// TIA Portal V19 export
FUNCTION_BLOCK "F_Zone25_FB"   // FB169, F_LAD
TITLE = SAFETY ZONE 25 - AREA 03 (PAREGGIAMENTO)
// stored: Access Published
   VAR
      D25 : "Door_FB";
      D27 : "Door_FB";
      FNS : "ForceNormalStop";
      F_Sinamics_Rulliera_1 : "FDevice_Sinamics_FB";
      F_Sinamics_Rulliera_2 : "FDevice_Sinamics_FB";
      F_Sinamics_PareggiatoreTesta : "FDevice_Sinamics_FB";
      F_Sinamics_PareggiatoreCoda : "FDevice_Sinamics_FB";
      F_Sinamics_ManipolatoreTesta : "FDevice_Sinamics_FB";
      F_Sinamics_ManipolatoreCoda : "FDevice_Sinamics_FB";
      F_Contactor_Valvole_Pareggiatore_Testa : "FDevice_Contactor_FB";
      F_Contactor_Valvole_Pareggiatore_Coda : "FDevice_Contactor_FB";
      F_Contactor_HU_CYTROPAC_STO { ExternalAccessible := 'False'; ExternalVisible := 'False'; ExternalWritable := 'False'} : "FDevice_Contactor_FB";
   END_VAR
   VAR_TEMP
      DoorNormalStop : Bool;
      DoorSafeStop : Bool;
      Door_Ok : Bool;
      FDBK : Bool;
   END_VAR
BEGIN

REGION Network 1: < < < < < < < < < < DOOR > > > > > > > > > >
END_REGION

REGION Network 2: Zone Entry enable
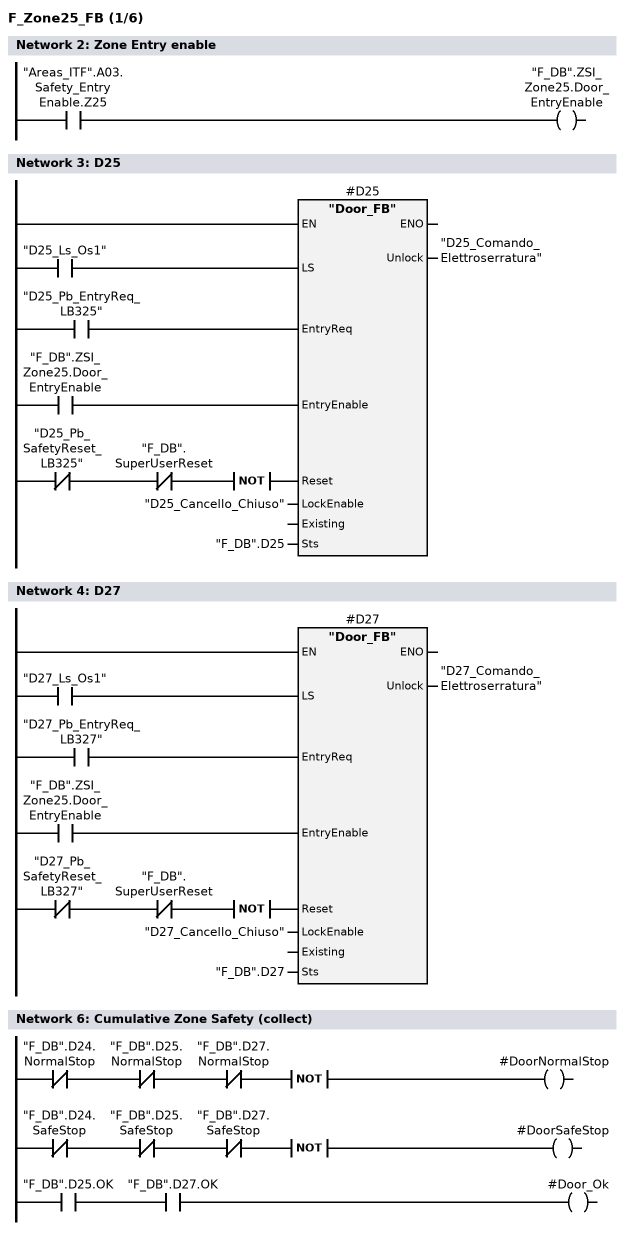
   RUNG wire#powerrail
      Contact( "Areas_ITF".A03.Safety_EntryEnable.Z25 )
      Coil( "F_DB".ZSI_Zone25.Door_EntryEnable )
   END_RUNG
   // the same network as SCL:
   "F_DB".ZSI_Zone25.Door_EntryEnable := "Areas_ITF".A03.Safety_EntryEnable.Z25;
END_REGION

REGION Network 3: D25
   RUNG wire#powerrail
      #D25(LS := wire#w1, EntryReq := wire#w2, EntryEnable := wire#w3, Reset := wire#w4, LockEnable := "D25_Cancello_Chiuso", Existing :=, Sts := "F_DB".D25, Unlock => "D25_Comando_Elettroserratura")
   END_RUNG
   RUNG wire#powerrail
      Contact( "D25_Ls_Os1" )
   END_RUNG wire#w1
   RUNG wire#powerrail
      Contact( "D25_Pb_EntryReq_LB325" )
   END_RUNG wire#w2
   RUNG wire#powerrail
      Contact( "F_DB".ZSI_Zone25.Door_EntryEnable )
   END_RUNG wire#w3
   RUNG wire#powerrail
      I_Contact( "D25_Pb_SafetyReset_LB325" )
      I_Contact( "F_DB".SuperUserReset )
      Not()
   END_RUNG wire#w4
   // the same network as SCL:
   #D25(LS := "D25_Ls_Os1",   // "Door_FB"
        EntryReq := "D25_Pb_EntryReq_LB325",
        EntryEnable := "F_DB".ZSI_Zone25.Door_EntryEnable,
        Reset := NOT (NOT "D25_Pb_SafetyReset_LB325" AND NOT "F_DB".SuperUserReset),
        LockEnable := "D25_Cancello_Chiuso",
        Sts := "F_DB".D25,
        Unlock => "D25_Comando_Elettroserratura");
END_REGION

REGION Network 4: D27
   RUNG wire#powerrail
      #D27(LS := wire#w1, EntryReq := wire#w2, EntryEnable := wire#w3, Reset := wire#w4, LockEnable := "D27_Cancello_Chiuso", Existing :=, Sts := "F_DB".D27, Unlock => "D27_Comando_Elettroserratura")
   END_RUNG
   RUNG wire#powerrail
      Contact( "D27_Ls_Os1" )
   END_RUNG wire#w1
   RUNG wire#powerrail
      Contact( "D27_Pb_EntryReq_LB327" )
   END_RUNG wire#w2
   RUNG wire#powerrail
      Contact( "F_DB".ZSI_Zone25.Door_EntryEnable )
   END_RUNG wire#w3
   RUNG wire#powerrail
      I_Contact( "D27_Pb_SafetyReset_LB327" )
      I_Contact( "F_DB".SuperUserReset )
      Not()
   END_RUNG wire#w4
   // the same network as SCL:
   #D27(LS := "D27_Ls_Os1",   // "Door_FB"
        EntryReq := "D27_Pb_EntryReq_LB327",
        EntryEnable := "F_DB".ZSI_Zone25.Door_EntryEnable,
        Reset := NOT (NOT "D27_Pb_SafetyReset_LB327" AND NOT "F_DB".SuperUserReset),
        LockEnable := "D27_Cancello_Chiuso",
        Sts := "F_DB".D27,
        Unlock => "D27_Comando_Elettroserratura");
END_REGION

REGION Network 5: < < < < < < < < < < ZONE SAFETY INTERFACE > > > > > > > > > >
END_REGION

REGION Network 6: Cumulative Zone Safety (collect)
   RUNG wire#powerrail
      I_Contact( "F_DB".D24.NormalStop )
      I_Contact( "F_DB".D25.NormalStop )
      I_Contact( "F_DB".D27.NormalStop )
      Not()
      Coil( #DoorNormalStop )
   END_RUNG
   RUNG wire#powerrail
      I_Contact( "F_DB".D24.SafeStop )
      I_Contact( "F_DB".D25.SafeStop )
      I_Contact( "F_DB".D27.SafeStop )
      Not()
      Coil( #DoorSafeStop )
   END_RUNG
   RUNG wire#powerrail
      Contact( "F_DB".D25.OK )
      Contact( "F_DB".D27.OK )
      Coil( #Door_Ok )
   END_RUNG
   // the same network as SCL:
   #DoorNormalStop := NOT (NOT "F_DB".D24.NormalStop AND NOT "F_DB".D25.NormalStop AND NOT "F_DB".D27.NormalStop);
   #DoorSafeStop := NOT (NOT "F_DB".D24.SafeStop AND NOT "F_DB".D25.SafeStop AND NOT "F_DB".D27.SafeStop);
   #Door_Ok := "F_DB".D25.OK AND "F_DB".D27.OK;
END_REGION

REGION Network 7: Zone must stay in Normal Stop During Restart
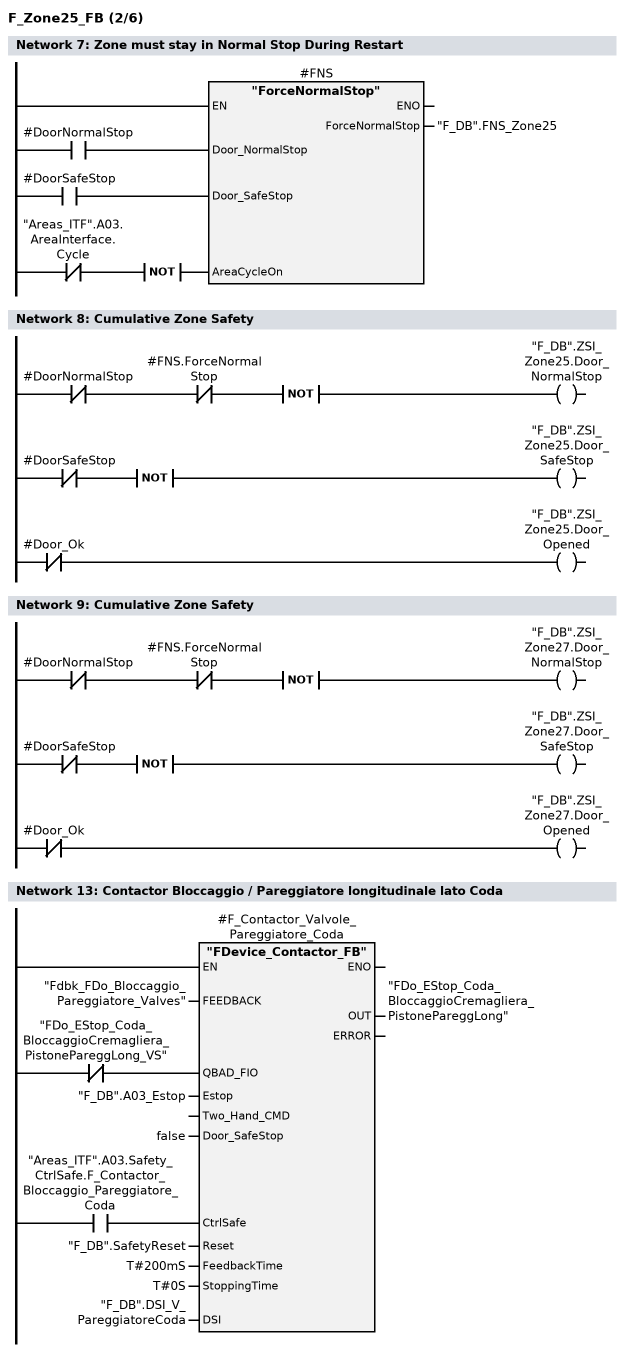
   RUNG wire#powerrail
      #FNS(Door_NormalStop := wire#w1, Door_SafeStop := wire#w2, AreaCycleOn := wire#w3, ForceNormalStop => "F_DB".FNS_Zone25)
   END_RUNG
   RUNG wire#powerrail
      Contact( #DoorNormalStop )
   END_RUNG wire#w1
   RUNG wire#powerrail
      Contact( #DoorSafeStop )
   END_RUNG wire#w2
   RUNG wire#powerrail
      I_Contact( "Areas_ITF".A03.AreaInterface.Cycle )
      Not()
   END_RUNG wire#w3
   // the same network as SCL:
   #FNS(Door_NormalStop := #DoorNormalStop,   // "ForceNormalStop"
        Door_SafeStop := #DoorSafeStop,
        AreaCycleOn := NOT (NOT "Areas_ITF".A03.AreaInterface.Cycle),
        ForceNormalStop => "F_DB".FNS_Zone25);
END_REGION

REGION Network 8: Cumulative Zone Safety
   RUNG wire#powerrail
      I_Contact( #DoorNormalStop )
      I_Contact( #FNS.ForceNormalStop )
      Not()
      Coil( "F_DB".ZSI_Zone25.Door_NormalStop )
   END_RUNG
   RUNG wire#powerrail
      I_Contact( #DoorSafeStop )
      Not()
      Coil( "F_DB".ZSI_Zone25.Door_SafeStop )
   END_RUNG
   RUNG wire#powerrail
      I_Contact( #Door_Ok )
      Coil( "F_DB".ZSI_Zone25.Door_Opened )
   END_RUNG
   // the same network as SCL:
   "F_DB".ZSI_Zone25.Door_NormalStop := NOT (NOT #DoorNormalStop AND NOT #FNS.ForceNormalStop);
   "F_DB".ZSI_Zone25.Door_SafeStop := NOT (NOT #DoorSafeStop);
   "F_DB".ZSI_Zone25.Door_Opened := NOT #Door_Ok;
END_REGION

REGION Network 9: Cumulative Zone Safety
   RUNG wire#powerrail
      I_Contact( #DoorNormalStop )
      I_Contact( #FNS.ForceNormalStop )
      Not()
      Coil( "F_DB".ZSI_Zone27.Door_NormalStop )
   END_RUNG
   RUNG wire#powerrail
      I_Contact( #DoorSafeStop )
      Not()
      Coil( "F_DB".ZSI_Zone27.Door_SafeStop )
   END_RUNG
   RUNG wire#powerrail
      I_Contact( #Door_Ok )
      Coil( "F_DB".ZSI_Zone27.Door_Opened )
   END_RUNG
   // the same network as SCL:
   "F_DB".ZSI_Zone27.Door_NormalStop := NOT (NOT #DoorNormalStop AND NOT #FNS.ForceNormalStop);
   "F_DB".ZSI_Zone27.Door_SafeStop := NOT (NOT #DoorSafeStop);
   "F_DB".ZSI_Zone27.Door_Opened := NOT #Door_Ok;
END_REGION

REGION Network 10: >
END_REGION

REGION Network 11: >
END_REGION

REGION Network 12: < < < < < < < < < < DEVICES SAFETY VALVES > > > > > > > > > >
END_REGION

REGION Network 13: Contactor Bloccaggio / Pareggiatore longitudinale lato Coda
   RUNG wire#powerrail
      #F_Contactor_Valvole_Pareggiatore_Coda(QBAD_FIO := wire#w1, CtrlSafe := wire#w2, FEEDBACK := "Fdbk_FDo_Bloccaggio_Pareggiatore_Valves", Estop := "F_DB".A03_Estop, Two_Hand_CMD :=, Door_SafeStop := false, Reset := "F_DB".SafetyReset, FeedbackTime := T#200mS, StoppingTime := T#0S, DSI := "F_DB".DSI_V_PareggiatoreCoda, OUT => "FDo_EStop_Coda_BloccaggioCremagliera_PistonePareggLong", ERROR =>)
   END_RUNG
   RUNG wire#powerrail
      I_Contact( "FDo_EStop_Coda_BloccaggioCremagliera_PistonePareggLong_VS" )
   END_RUNG wire#w1
   RUNG wire#powerrail
      Contact( "Areas_ITF".A03.Safety_CtrlSafe.F_Contactor_Bloccaggio_Pareggiatore_Coda )
   END_RUNG wire#w2
   // the same network as SCL:
   #F_Contactor_Valvole_Pareggiatore_Coda(FEEDBACK := "Fdbk_FDo_Bloccaggio_Pareggiatore_Valves",   // "FDevice_Contactor_FB"
                           QBAD_FIO := NOT "FDo_EStop_Coda_BloccaggioCremagliera_PistonePareggLong_VS",
                           Estop := "F_DB".A03_Estop,
                           Door_SafeStop := false,
                           CtrlSafe := "Areas_ITF".A03.Safety_CtrlSafe.F_Contactor_Bloccaggio_Pareggiatore_Coda,
                           Reset := "F_DB".SafetyReset,
                           FeedbackTime := T#200mS,
                           StoppingTime := T#0S,
                           DSI := "F_DB".DSI_V_PareggiatoreCoda,
                           OUT => "FDo_EStop_Coda_BloccaggioCremagliera_PistonePareggLong");
END_REGION

REGION Network 14: Contactor Bloccaggio lato testa
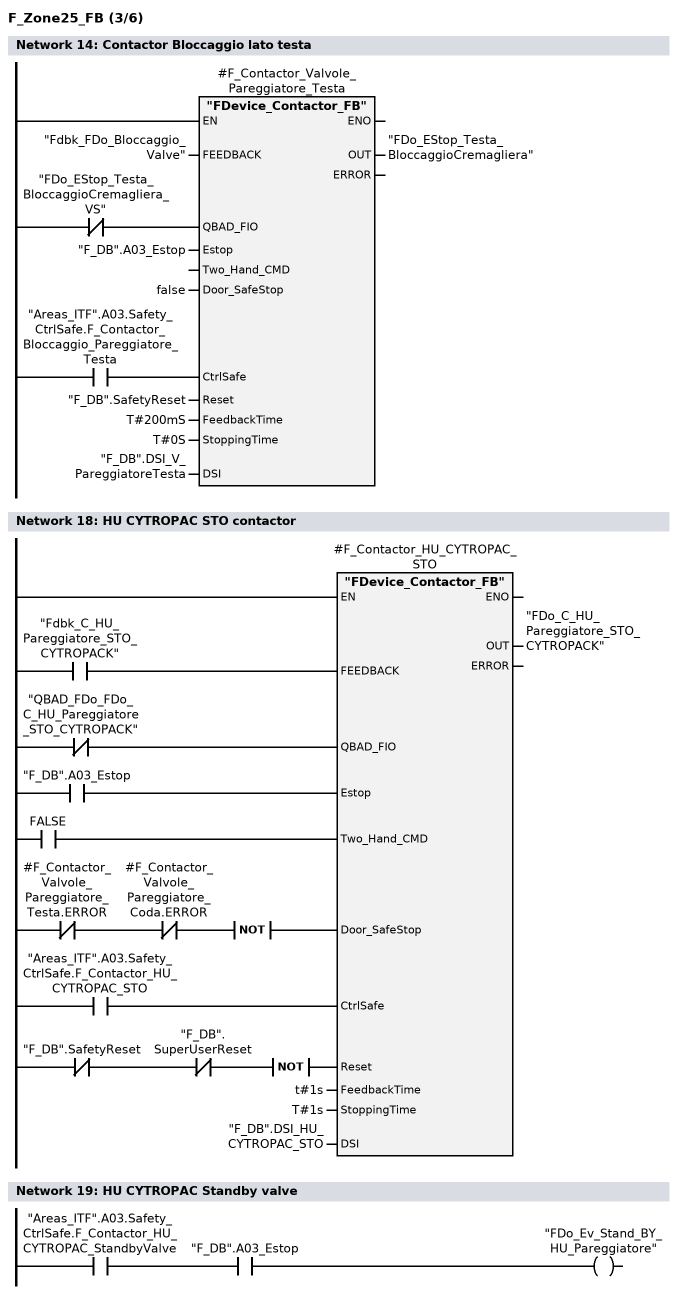
   RUNG wire#powerrail
      #F_Contactor_Valvole_Pareggiatore_Testa(QBAD_FIO := wire#w1, CtrlSafe := wire#w2, FEEDBACK := "Fdbk_FDo_Bloccaggio_Valve", Estop := "F_DB".A03_Estop, Two_Hand_CMD :=, Door_SafeStop := false, Reset := "F_DB".SafetyReset, FeedbackTime := T#200mS, StoppingTime := T#0S, DSI := "F_DB".DSI_V_PareggiatoreTesta, OUT => "FDo_EStop_Testa_BloccaggioCremagliera", ERROR =>)
   END_RUNG
   RUNG wire#powerrail
      I_Contact( "FDo_EStop_Testa_BloccaggioCremagliera_VS" )
   END_RUNG wire#w1
   RUNG wire#powerrail
      Contact( "Areas_ITF".A03.Safety_CtrlSafe.F_Contactor_Bloccaggio_Pareggiatore_Testa )
   END_RUNG wire#w2
   // the same network as SCL:
   #F_Contactor_Valvole_Pareggiatore_Testa(FEEDBACK := "Fdbk_FDo_Bloccaggio_Valve",   // "FDevice_Contactor_FB"
                           QBAD_FIO := NOT "FDo_EStop_Testa_BloccaggioCremagliera_VS",
                           Estop := "F_DB".A03_Estop,
                           Door_SafeStop := false,
                           CtrlSafe := "Areas_ITF".A03.Safety_CtrlSafe.F_Contactor_Bloccaggio_Pareggiatore_Testa,
                           Reset := "F_DB".SafetyReset,
                           FeedbackTime := T#200mS,
                           StoppingTime := T#0S,
                           DSI := "F_DB".DSI_V_PareggiatoreTesta,
                           OUT => "FDo_EStop_Testa_BloccaggioCremagliera");
END_REGION

REGION Network 15: >
END_REGION

REGION Network 16: >
END_REGION

REGION Network 17: < < < < < < < < < < DEVICES CONTACTORS > > > > > > > > > >
END_REGION

REGION Network 18: HU CYTROPAC STO contactor
   RUNG wire#powerrail
      #F_Contactor_HU_CYTROPAC_STO(FEEDBACK := wire#w1, QBAD_FIO := wire#w2, Estop := wire#w3, Two_Hand_CMD := wire#w4, Door_SafeStop := wire#w5, CtrlSafe := wire#w6, Reset := wire#w7, FeedbackTime := t#1s, StoppingTime := T#1s, DSI := "F_DB".DSI_HU_CYTROPAC_STO, OUT => "FDo_C_HU_Pareggiatore_STO_CYTROPACK", ERROR =>)
   END_RUNG
   RUNG wire#powerrail
      Contact( "Fdbk_C_HU_Pareggiatore_STO_CYTROPACK" )
   END_RUNG wire#w1
   RUNG wire#powerrail
      I_Contact( "QBAD_FDo_FDo_C_HU_Pareggiatore_STO_CYTROPACK" )
   END_RUNG wire#w2
   RUNG wire#powerrail
      Contact( "F_DB".A03_Estop )
   END_RUNG wire#w3
   RUNG wire#powerrail
      Contact( FALSE )
   END_RUNG wire#w4
   RUNG wire#powerrail
      I_Contact( #F_Contactor_Valvole_Pareggiatore_Testa.ERROR )
      I_Contact( #F_Contactor_Valvole_Pareggiatore_Coda.ERROR )
      Not()
   END_RUNG wire#w5
   RUNG wire#powerrail
      Contact( "Areas_ITF".A03.Safety_CtrlSafe.F_Contactor_HU_CYTROPAC_STO )
   END_RUNG wire#w6
   RUNG wire#powerrail
      I_Contact( "F_DB".SafetyReset )
      I_Contact( "F_DB".SuperUserReset )
      Not()
   END_RUNG wire#w7
   // the same network as SCL:
   #F_Contactor_HU_CYTROPAC_STO(FEEDBACK := "Fdbk_C_HU_Pareggiatore_STO_CYTROPACK",   // "FDevice_Contactor_FB"
                           QBAD_FIO := NOT "QBAD_FDo_FDo_C_HU_Pareggiatore_STO_CYTROPACK",
                           Estop := "F_DB".A03_Estop,
                           Two_Hand_CMD := FALSE,
                           Door_SafeStop := NOT (NOT #F_Contactor_Valvole_Pareggiatore_Testa.ERROR AND NOT #F_Contactor_Valvole_Pareggiatore_Coda.ERROR),
                           CtrlSafe := "Areas_ITF".A03.Safety_CtrlSafe.F_Contactor_HU_CYTROPAC_STO,
                           Reset := NOT (NOT "F_DB".SafetyReset AND NOT "F_DB".SuperUserReset),
                           FeedbackTime := t#1s,
                           StoppingTime := T#1s,
                           DSI := "F_DB".DSI_HU_CYTROPAC_STO,
                           OUT => "FDo_C_HU_Pareggiatore_STO_CYTROPACK");
END_REGION

REGION Network 19: HU CYTROPAC Standby valve
   RUNG wire#powerrail
      Contact( "Areas_ITF".A03.Safety_CtrlSafe.F_Contactor_HU_CYTROPAC_StandbyValve )
      Contact( "F_DB".A03_Estop )
      Coil( "FDo_Ev_Stand_BY_HU_Pareggiatore" )
   END_RUNG
   // the same network as SCL:
   "FDo_Ev_Stand_BY_HU_Pareggiatore" := "Areas_ITF".A03.Safety_CtrlSafe.F_Contactor_HU_CYTROPAC_StandbyValve AND "F_DB".A03_Estop;
END_REGION

REGION Network 20: >
END_REGION

REGION Network 21: >
END_REGION

REGION Network 22: < < < < < < < < < < DEVICES S120 > > > > > > > > > >
END_REGION

REGION Network 23: S120 - Ax Rulliera 1
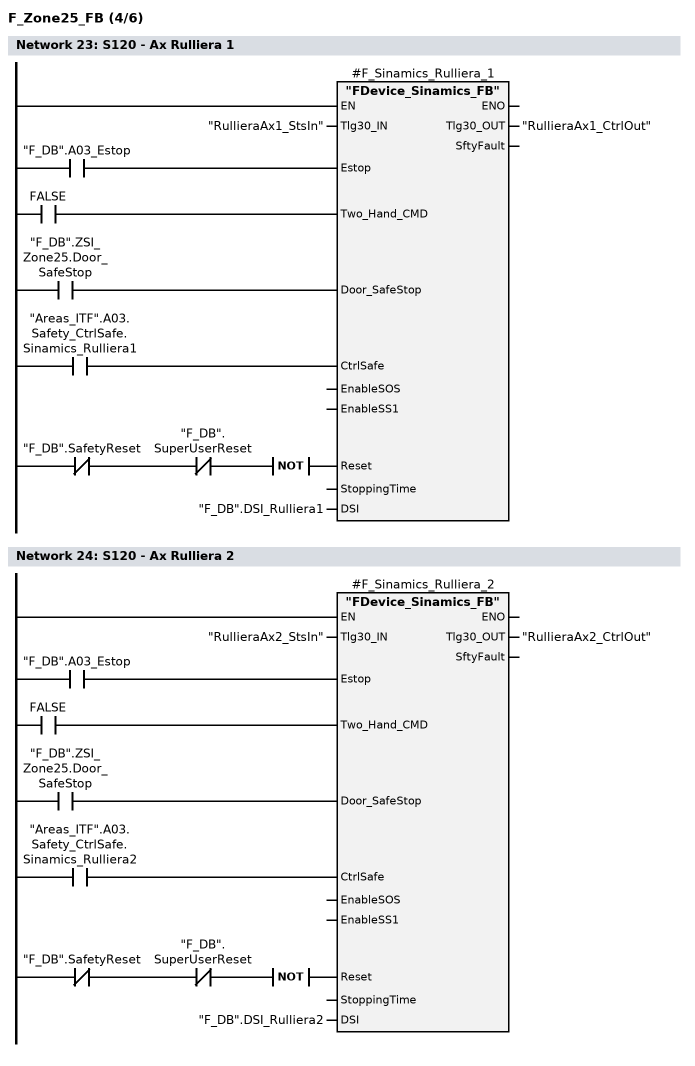
   RUNG wire#powerrail
      #F_Sinamics_Rulliera_1(Estop := wire#w1, Two_Hand_CMD := wire#w2, Door_SafeStop := wire#w3, CtrlSafe := wire#w4, Reset := wire#w5, Tlg30_IN := "RullieraAx1_StsIn", EnableSOS :=, EnableSS1 :=, StoppingTime :=, DSI := "F_DB".DSI_Rulliera1, Tlg30_OUT => "RullieraAx1_CtrlOut", SftyFault =>)
   END_RUNG
   RUNG wire#powerrail
      Contact( "F_DB".A03_Estop )
   END_RUNG wire#w1
   RUNG wire#powerrail
      Contact( FALSE )
   END_RUNG wire#w2
   RUNG wire#powerrail
      Contact( "F_DB".ZSI_Zone25.Door_SafeStop )
   END_RUNG wire#w3
   RUNG wire#powerrail
      Contact( "Areas_ITF".A03.Safety_CtrlSafe.Sinamics_Rulliera1 )
   END_RUNG wire#w4
   RUNG wire#powerrail
      I_Contact( "F_DB".SafetyReset )
      I_Contact( "F_DB".SuperUserReset )
      Not()
   END_RUNG wire#w5
   // the same network as SCL:
   #F_Sinamics_Rulliera_1(Tlg30_IN := "RullieraAx1_StsIn",   // "FDevice_Sinamics_FB"
                          Estop := "F_DB".A03_Estop,
                          Two_Hand_CMD := FALSE,
                          Door_SafeStop := "F_DB".ZSI_Zone25.Door_SafeStop,
                          CtrlSafe := "Areas_ITF".A03.Safety_CtrlSafe.Sinamics_Rulliera1,
                          Reset := NOT (NOT "F_DB".SafetyReset AND NOT "F_DB".SuperUserReset),
                          DSI := "F_DB".DSI_Rulliera1,
                          Tlg30_OUT => "RullieraAx1_CtrlOut");
END_REGION

REGION Network 24: S120 - Ax Rulliera 2
   RUNG wire#powerrail
      #F_Sinamics_Rulliera_2(Estop := wire#w1, Two_Hand_CMD := wire#w2, Door_SafeStop := wire#w3, CtrlSafe := wire#w4, Reset := wire#w5, Tlg30_IN := "RullieraAx2_StsIn", EnableSOS :=, EnableSS1 :=, StoppingTime :=, DSI := "F_DB".DSI_Rulliera2, Tlg30_OUT => "RullieraAx2_CtrlOut", SftyFault =>)
   END_RUNG
   RUNG wire#powerrail
      Contact( "F_DB".A03_Estop )
   END_RUNG wire#w1
   RUNG wire#powerrail
      Contact( FALSE )
   END_RUNG wire#w2
   RUNG wire#powerrail
      Contact( "F_DB".ZSI_Zone25.Door_SafeStop )
   END_RUNG wire#w3
   RUNG wire#powerrail
      Contact( "Areas_ITF".A03.Safety_CtrlSafe.Sinamics_Rulliera2 )
   END_RUNG wire#w4
   RUNG wire#powerrail
      I_Contact( "F_DB".SafetyReset )
      I_Contact( "F_DB".SuperUserReset )
      Not()
   END_RUNG wire#w5
   // the same network as SCL:
   #F_Sinamics_Rulliera_2(Tlg30_IN := "RullieraAx2_StsIn",   // "FDevice_Sinamics_FB"
                          Estop := "F_DB".A03_Estop,
                          Two_Hand_CMD := FALSE,
                          Door_SafeStop := "F_DB".ZSI_Zone25.Door_SafeStop,
                          CtrlSafe := "Areas_ITF".A03.Safety_CtrlSafe.Sinamics_Rulliera2,
                          Reset := NOT (NOT "F_DB".SafetyReset AND NOT "F_DB".SuperUserReset),
                          DSI := "F_DB".DSI_Rulliera2,
                          Tlg30_OUT => "RullieraAx2_CtrlOut");
END_REGION

REGION Network 25: S120 - Ax Pareggiatore Testa
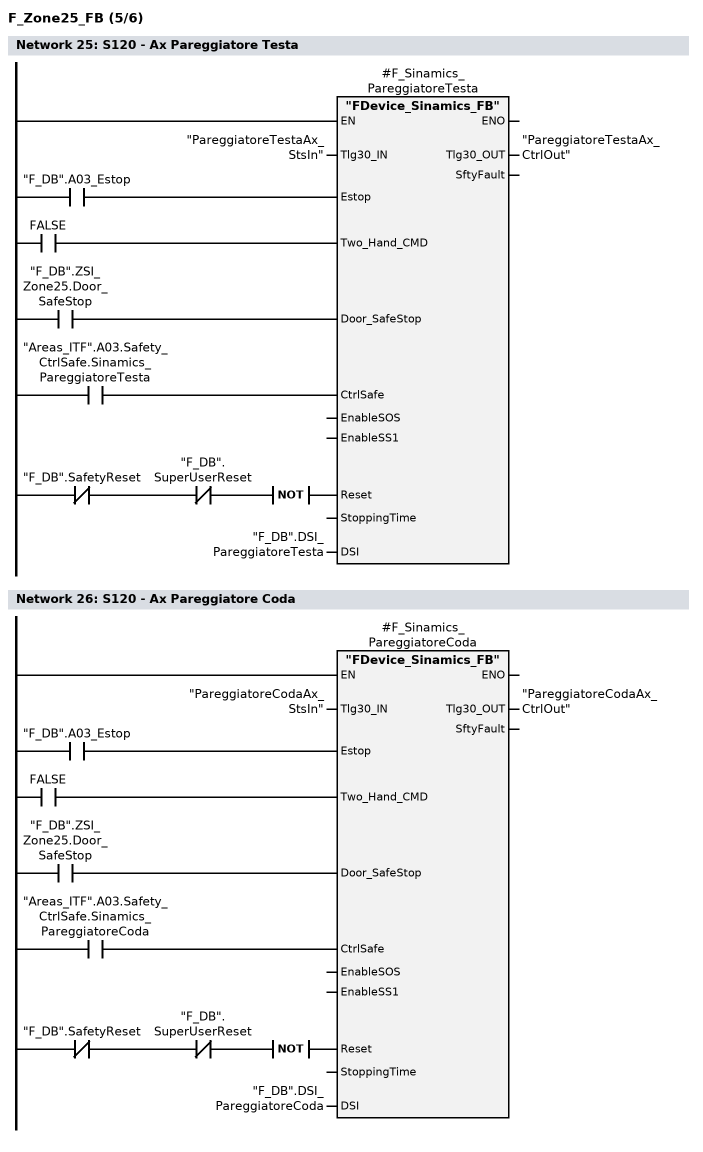
   RUNG wire#powerrail
      #F_Sinamics_PareggiatoreTesta(Estop := wire#w1, Two_Hand_CMD := wire#w2, Door_SafeStop := wire#w3, CtrlSafe := wire#w4, Reset := wire#w5, Tlg30_IN := "PareggiatoreTestaAx_StsIn", EnableSOS :=, EnableSS1 :=, StoppingTime :=, DSI := "F_DB".DSI_PareggiatoreTesta, Tlg30_OUT => "PareggiatoreTestaAx_CtrlOut", SftyFault =>)
   END_RUNG
   RUNG wire#powerrail
      Contact( "F_DB".A03_Estop )
   END_RUNG wire#w1
   RUNG wire#powerrail
      Contact( FALSE )
   END_RUNG wire#w2
   RUNG wire#powerrail
      Contact( "F_DB".ZSI_Zone25.Door_SafeStop )
   END_RUNG wire#w3
   RUNG wire#powerrail
      Contact( "Areas_ITF".A03.Safety_CtrlSafe.Sinamics_PareggiatoreTesta )
   END_RUNG wire#w4
   RUNG wire#powerrail
      I_Contact( "F_DB".SafetyReset )
      I_Contact( "F_DB".SuperUserReset )
      Not()
   END_RUNG wire#w5
   // the same network as SCL:
   #F_Sinamics_PareggiatoreTesta(Tlg30_IN := "PareggiatoreTestaAx_StsIn",   // "FDevice_Sinamics_FB"
                           Estop := "F_DB".A03_Estop,
                           Two_Hand_CMD := FALSE,
                           Door_SafeStop := "F_DB".ZSI_Zone25.Door_SafeStop,
                           CtrlSafe := "Areas_ITF".A03.Safety_CtrlSafe.Sinamics_PareggiatoreTesta,
                           Reset := NOT (NOT "F_DB".SafetyReset AND NOT "F_DB".SuperUserReset),
                           DSI := "F_DB".DSI_PareggiatoreTesta,
                           Tlg30_OUT => "PareggiatoreTestaAx_CtrlOut");
END_REGION

REGION Network 26: S120 - Ax Pareggiatore Coda
   RUNG wire#powerrail
      #F_Sinamics_PareggiatoreCoda(Estop := wire#w1, Two_Hand_CMD := wire#w2, Door_SafeStop := wire#w3, CtrlSafe := wire#w4, Reset := wire#w5, Tlg30_IN := "PareggiatoreCodaAx_StsIn", EnableSOS :=, EnableSS1 :=, StoppingTime :=, DSI := "F_DB".DSI_PareggiatoreCoda, Tlg30_OUT => "PareggiatoreCodaAx_CtrlOut", SftyFault =>)
   END_RUNG
   RUNG wire#powerrail
      Contact( "F_DB".A03_Estop )
   END_RUNG wire#w1
   RUNG wire#powerrail
      Contact( FALSE )
   END_RUNG wire#w2
   RUNG wire#powerrail
      Contact( "F_DB".ZSI_Zone25.Door_SafeStop )
   END_RUNG wire#w3
   RUNG wire#powerrail
      Contact( "Areas_ITF".A03.Safety_CtrlSafe.Sinamics_PareggiatoreCoda )
   END_RUNG wire#w4
   RUNG wire#powerrail
      I_Contact( "F_DB".SafetyReset )
      I_Contact( "F_DB".SuperUserReset )
      Not()
   END_RUNG wire#w5
   // the same network as SCL:
   #F_Sinamics_PareggiatoreCoda(Tlg30_IN := "PareggiatoreCodaAx_StsIn",   // "FDevice_Sinamics_FB"
                           Estop := "F_DB".A03_Estop,
                           Two_Hand_CMD := FALSE,
                           Door_SafeStop := "F_DB".ZSI_Zone25.Door_SafeStop,
                           CtrlSafe := "Areas_ITF".A03.Safety_CtrlSafe.Sinamics_PareggiatoreCoda,
                           Reset := NOT (NOT "F_DB".SafetyReset AND NOT "F_DB".SuperUserReset),
                           DSI := "F_DB".DSI_PareggiatoreCoda,
                           Tlg30_OUT => "PareggiatoreCodaAx_CtrlOut");
END_REGION

REGION Network 27: S120 - Ax Manipolatore Testa
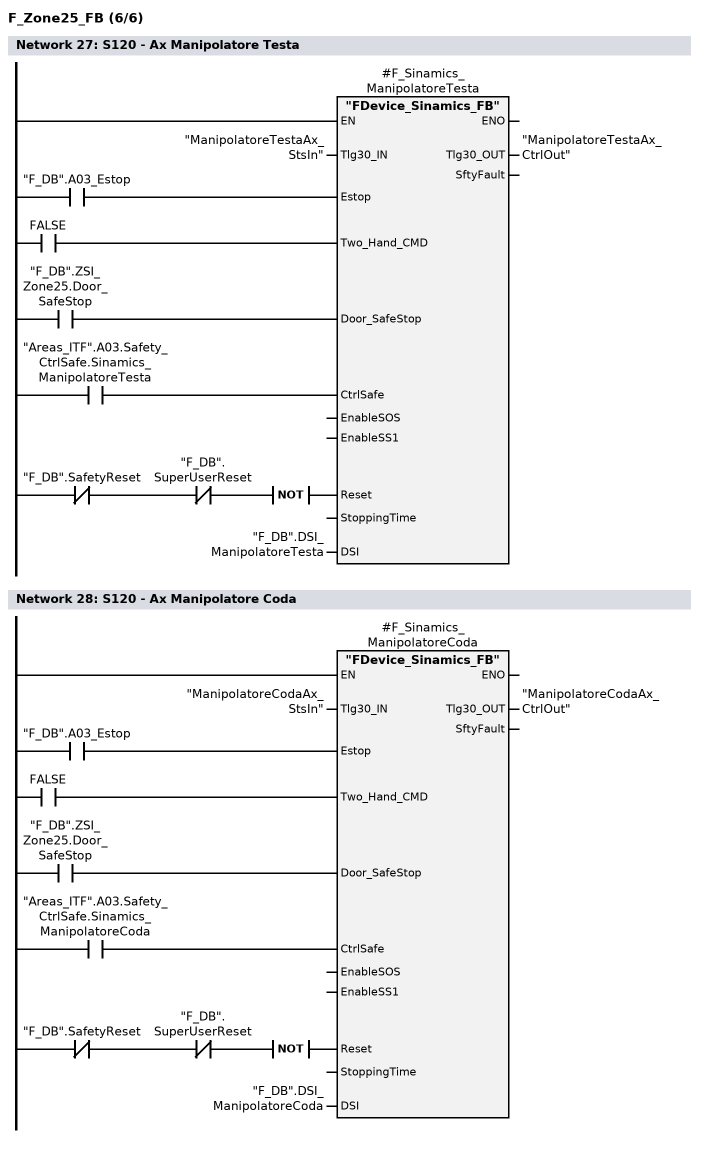
   RUNG wire#powerrail
      #F_Sinamics_ManipolatoreTesta(Estop := wire#w1, Two_Hand_CMD := wire#w2, Door_SafeStop := wire#w3, CtrlSafe := wire#w4, Reset := wire#w5, Tlg30_IN := "ManipolatoreTestaAx_StsIn", EnableSOS :=, EnableSS1 :=, StoppingTime :=, DSI := "F_DB".DSI_ManipolatoreTesta, Tlg30_OUT => "ManipolatoreTestaAx_CtrlOut", SftyFault =>)
   END_RUNG
   RUNG wire#powerrail
      Contact( "F_DB".A03_Estop )
   END_RUNG wire#w1
   RUNG wire#powerrail
      Contact( FALSE )
   END_RUNG wire#w2
   RUNG wire#powerrail
      Contact( "F_DB".ZSI_Zone25.Door_SafeStop )
   END_RUNG wire#w3
   RUNG wire#powerrail
      Contact( "Areas_ITF".A03.Safety_CtrlSafe.Sinamics_ManipolatoreTesta )
   END_RUNG wire#w4
   RUNG wire#powerrail
      I_Contact( "F_DB".SafetyReset )
      I_Contact( "F_DB".SuperUserReset )
      Not()
   END_RUNG wire#w5
   // the same network as SCL:
   #F_Sinamics_ManipolatoreTesta(Tlg30_IN := "ManipolatoreTestaAx_StsIn",   // "FDevice_Sinamics_FB"
                           Estop := "F_DB".A03_Estop,
                           Two_Hand_CMD := FALSE,
                           Door_SafeStop := "F_DB".ZSI_Zone25.Door_SafeStop,
                           CtrlSafe := "Areas_ITF".A03.Safety_CtrlSafe.Sinamics_ManipolatoreTesta,
                           Reset := NOT (NOT "F_DB".SafetyReset AND NOT "F_DB".SuperUserReset),
                           DSI := "F_DB".DSI_ManipolatoreTesta,
                           Tlg30_OUT => "ManipolatoreTestaAx_CtrlOut");
END_REGION

REGION Network 28: S120 - Ax Manipolatore Coda
   RUNG wire#powerrail
      #F_Sinamics_ManipolatoreCoda(Estop := wire#w1, Two_Hand_CMD := wire#w2, Door_SafeStop := wire#w3, CtrlSafe := wire#w4, Reset := wire#w5, Tlg30_IN := "ManipolatoreCodaAx_StsIn", EnableSOS :=, EnableSS1 :=, StoppingTime :=, DSI := "F_DB".DSI_ManipolatoreCoda, Tlg30_OUT => "ManipolatoreCodaAx_CtrlOut", SftyFault =>)
   END_RUNG
   RUNG wire#powerrail
      Contact( "F_DB".A03_Estop )
   END_RUNG wire#w1
   RUNG wire#powerrail
      Contact( FALSE )
   END_RUNG wire#w2
   RUNG wire#powerrail
      Contact( "F_DB".ZSI_Zone25.Door_SafeStop )
   END_RUNG wire#w3
   RUNG wire#powerrail
      Contact( "Areas_ITF".A03.Safety_CtrlSafe.Sinamics_ManipolatoreCoda )
   END_RUNG wire#w4
   RUNG wire#powerrail
      I_Contact( "F_DB".SafetyReset )
      I_Contact( "F_DB".SuperUserReset )
      Not()
   END_RUNG wire#w5
   // the same network as SCL:
   #F_Sinamics_ManipolatoreCoda(Tlg30_IN := "ManipolatoreCodaAx_StsIn",   // "FDevice_Sinamics_FB"
                           Estop := "F_DB".A03_Estop,
                           Two_Hand_CMD := FALSE,
                           Door_SafeStop := "F_DB".ZSI_Zone25.Door_SafeStop,
                           CtrlSafe := "Areas_ITF".A03.Safety_CtrlSafe.Sinamics_ManipolatoreCoda,
                           Reset := NOT (NOT "F_DB".SafetyReset AND NOT "F_DB".SuperUserReset),
                           DSI := "F_DB".DSI_ManipolatoreCoda,
                           Tlg30_OUT => "ManipolatoreCodaAx_CtrlOut");
END_REGION

REGION Network 29: >
END_REGION

REGION Network 30: >
END_REGION
END_FUNCTION_BLOCK
